// Mitsubishi GX Works2 project: PuyoPuyo_Ver100_20220530   PLC: Q03UDV

PROGRAM 11_DEBUG  // Test Function for Debug
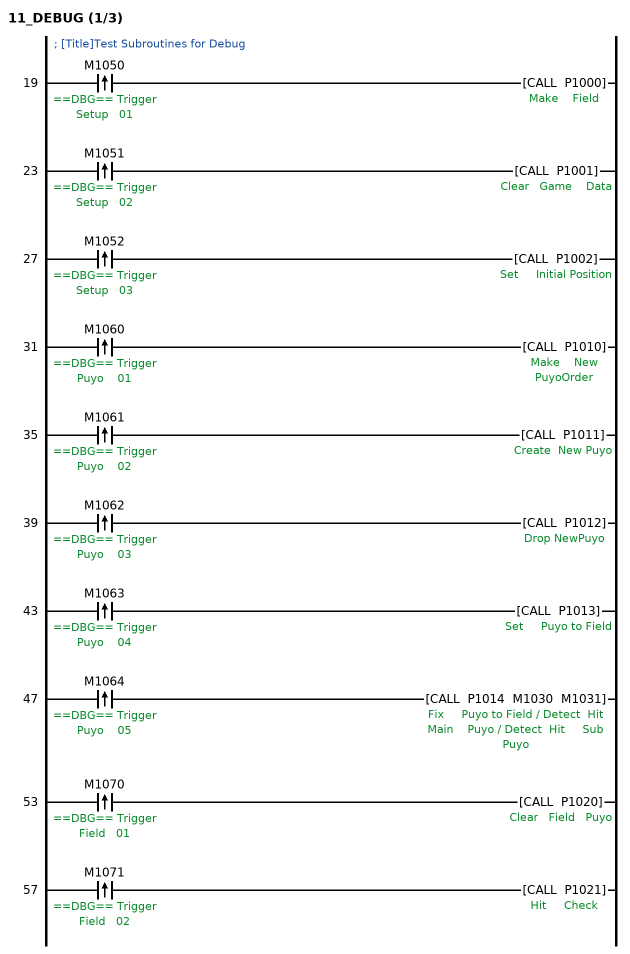
; [Title]Test Subroutines for Debug
19    LDP     M1050  ; ==DBG== Trigger Setup   01
      CALL    P1000  ; Make    Field
23    LDP     M1051  ; ==DBG== Trigger Setup   02
      CALL    P1001  ; Clear   Game    Data
27    LDP     M1052  ; ==DBG== Trigger Setup   03
      CALL    P1002  ; Set     Initial Position
31    LDP     M1060  ; ==DBG== Trigger Puyo    01
      CALL    P1010  ; Make    New PuyoOrder
35    LDP     M1061  ; ==DBG== Trigger Puyo    02
      CALL    P1011  ; Create  New Puyo
39    LDP     M1062  ; ==DBG== Trigger Puyo    03
      CALL    P1012  ; Drop NewPuyo
43    LDP     M1063  ; ==DBG== Trigger Puyo    04
      CALL    P1013  ; Set     Puyo to Field
47    LDP     M1064  ; ==DBG== Trigger Puyo    05
      CALL    P1014 M1030 M1031  ; Fix     Puyo to Field / Detect  Hit     Main    Puyo / Detect  Hit     Sub     Puyo
53    LDP     M1070  ; ==DBG== Trigger Field   01
      CALL    P1020  ; Clear   Field   Puyo
57    LDP     M1071  ; ==DBG== Trigger Field   02
      CALL    P1021  ; Hit     Check
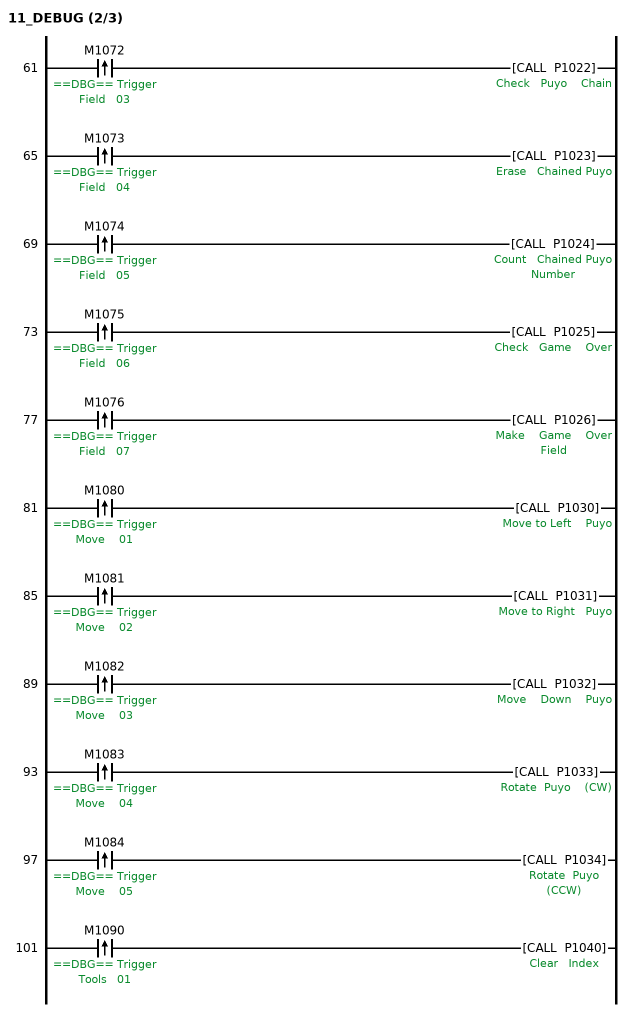
61    LDP     M1072  ; ==DBG== Trigger Field   03
      CALL    P1022  ; Check   Puyo    Chain
65    LDP     M1073  ; ==DBG== Trigger Field   04
      CALL    P1023  ; Erase   Chained Puyo
69    LDP     M1074  ; ==DBG== Trigger Field   05
      CALL    P1024  ; Count   Chained Puyo    Number
73    LDP     M1075  ; ==DBG== Trigger Field   06
      CALL    P1025  ; Check   Game    Over
77    LDP     M1076  ; ==DBG== Trigger Field   07
      CALL    P1026  ; Make    Game    Over    Field
81    LDP     M1080  ; ==DBG== Trigger Move    01
      CALL    P1030  ; Move to Left    Puyo
85    LDP     M1081  ; ==DBG== Trigger Move    02
      CALL    P1031  ; Move to Right   Puyo
89    LDP     M1082  ; ==DBG== Trigger Move    03
      CALL    P1032  ; Move    Down    Puyo
93    LDP     M1083  ; ==DBG== Trigger Move    04
      CALL    P1033  ; Rotate  Puyo    (CW)
97    LDP     M1084  ; ==DBG== Trigger Move    05
      CALL    P1034  ; Rotate  Puyo    (CCW)
101   LDP     M1090  ; ==DBG== Trigger Tools   01
      CALL    P1040  ; Clear   Index
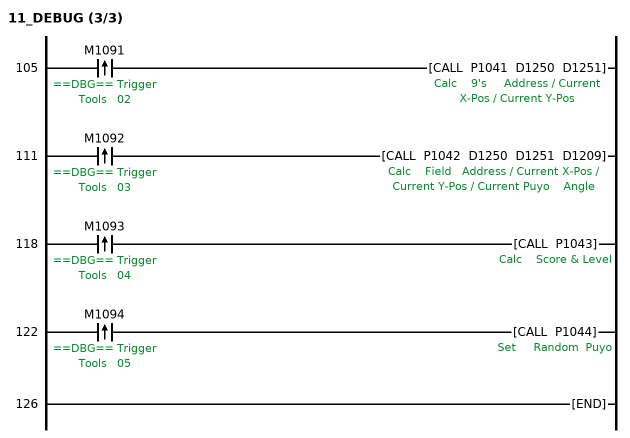
105   LDP     M1091  ; ==DBG== Trigger Tools   02
      CALL    P1041 D1250 D1251  ; Calc    9's     Address / Current X-Pos / Current Y-Pos
111   LDP     M1092  ; ==DBG== Trigger Tools   03
      CALL    P1042 D1250 D1251 D1209  ; Calc    Field   Address / Current Puyo    Angle
118   LDP     M1093  ; ==DBG== Trigger Tools   04
      CALL    P1043  ; Calc    Score & Level
122   LDP     M1094  ; ==DBG== Trigger Tools   05
      CALL    P1044  ; Set     Random  Puyo
126   END
END_PROGRAM

PROGRAM 95_TOOL  // Common Tools
; [Title]P1040 Clear Index
      P1040
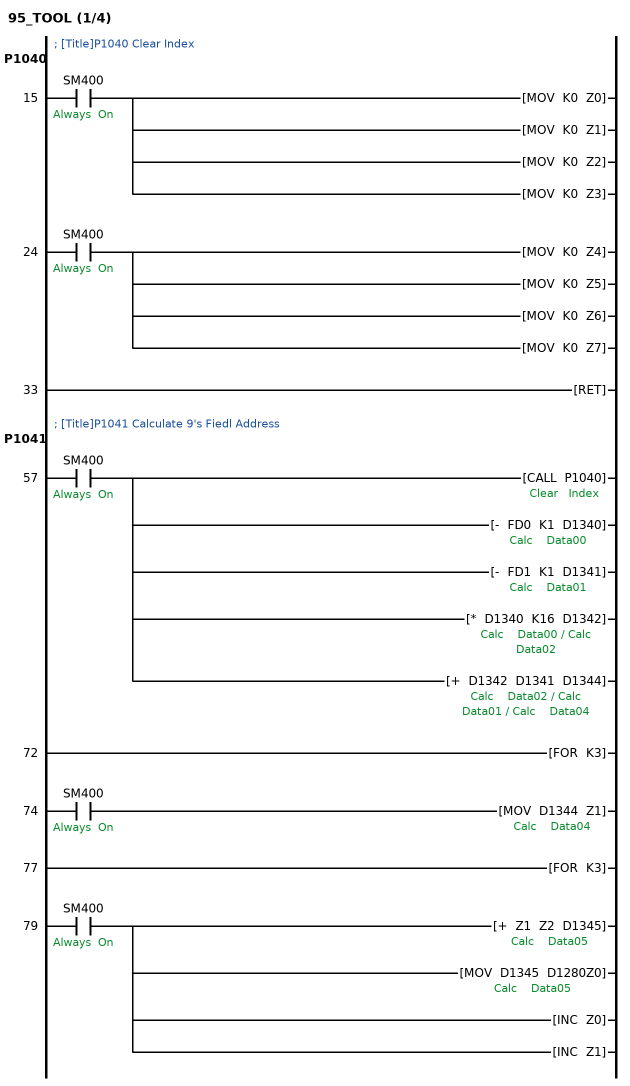
15    LD      SM400  ; Always  On
      MOV     K0 Z0
      MOV     K0 Z1
      MOV     K0 Z2
      MOV     K0 Z3
24    LD      SM400  ; Always  On
      MOV     K0 Z4
      MOV     K0 Z5
      MOV     K0 Z6
      MOV     K0 Z7
33    RET
; [Title]P1041 Calculate 9's Fiedl Address
      P1041
57    LD      SM400  ; Always  On
      CALL    P1040  ; Clear   Index
      -       FD0 K1 D1340  ; Calc    Data00
      -       FD1 K1 D1341  ; Calc    Data01
      *       D1340 K16 D1342  ; Calc    Data02
      +       D1342 D1341 D1344  ; Calc    Data04
72    FOR     K3
74    LD      SM400  ; Always  On
      MOV     D1344 Z1
77    FOR     K3
79    LD      SM400  ; Always  On
      +       Z1 Z2 D1345  ; Calc    Data05
      MOV     D1345 D1280Z0
      INC     Z0
      INC     Z1
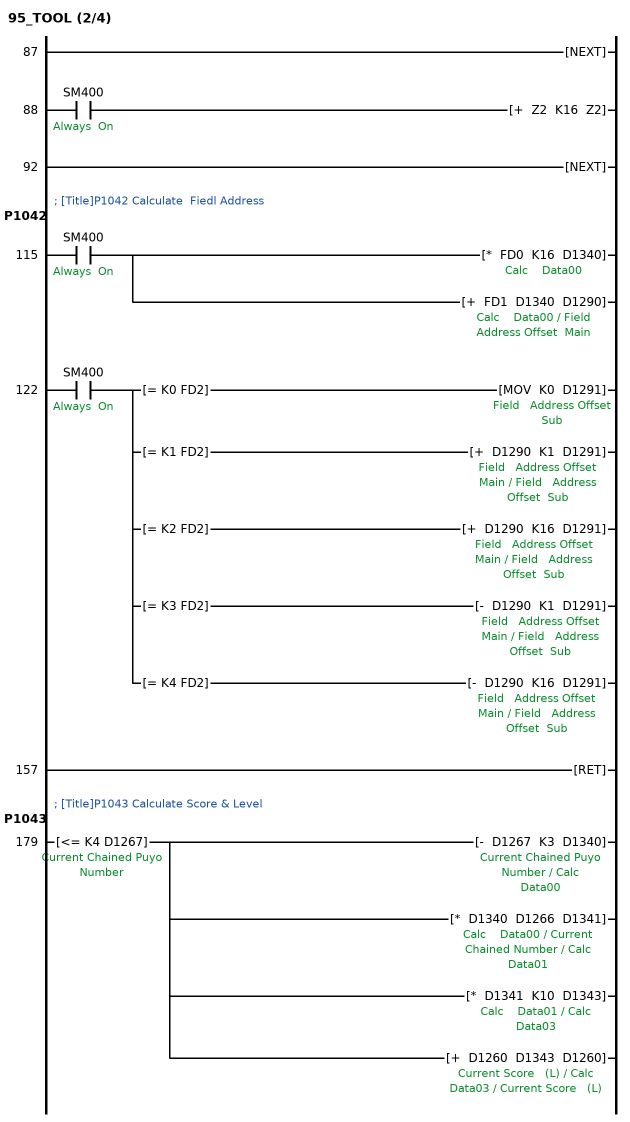
87    NEXT
88    LD      SM400  ; Always  On
      +       Z2 K16 Z2
92    NEXT
; [Title]P1042 Calculate  Fiedl Address
      P1042
115   LD      SM400  ; Always  On
      *       FD0 K16 D1340
      +       FD1 D1340 D1290  ; Field   Address Offset  Main
122   LD      SM400  ; Always  On
      MPS
      AND=    K0 FD2
      MOV     K0 D1291  ; Field   Address Offset  Sub
      MRD
      AND=    K1 FD2
      +       D1290 K1 D1291
      MRD
      AND=    K2 FD2
      +       D1290 K16 D1291
      MRD
      AND=    K3 FD2
      -       D1290 K1 D1291
      MPP
      AND=    K4 FD2
      -       D1290 K16 D1291
157   RET
; [Title]P1043 Calculate Score & Level
      P1043
179   LD<=    K4 D1267  ; Current Chained Puyo    Number
      -       D1267 K3 D1340
      *       D1340 D1266 D1341  ; Current Chained Number
      *       D1341 K10 D1343  ; Calc    Data03
      +       D1260 D1343 D1260  ; Current Score   (L)
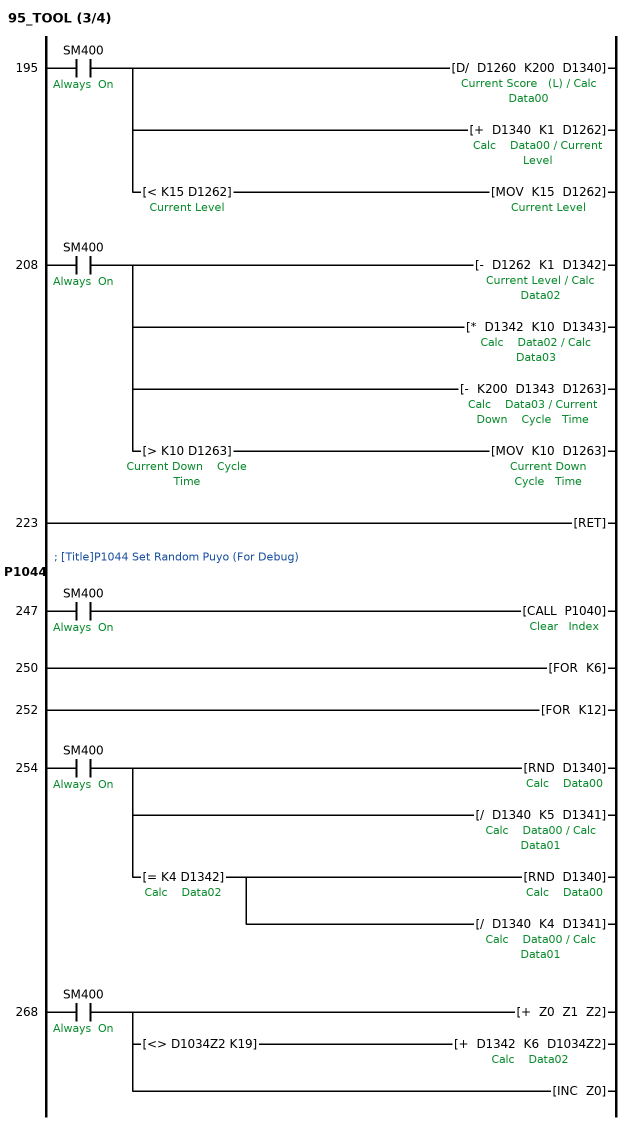
195   LD      SM400  ; Always  On
      D/      D1260 K200 D1340
      +       D1340 K1 D1262  ; Current Level
      AND<    K15 D1262  ; Current Level
      MOV     K15 D1262
208   LD      SM400  ; Always  On
      -       D1262 K1 D1342
      *       D1342 K10 D1343
      -       K200 D1343 D1263  ; Current Down    Cycle   Time
      AND>    K10 D1263  ; Current Down    Cycle   Time
      MOV     K10 D1263
223   RET
; [Title]P1044 Set Random Puyo (For Debug)
      P1044
247   LD      SM400  ; Always  On
      CALL    P1040
250   FOR     K6
252   FOR     K12
254   LD      SM400  ; Always  On
      RND     D1340
      /       D1340 K5 D1341
      AND=    K4 D1342  ; Calc    Data02
      RND     D1340
      /       D1340 K4 D1341
268   LD      SM400  ; Always  On
      +       Z0 Z1 Z2
      MPS
      AND<>   D1034Z2 K19
      +       D1342 K6 D1034Z2
      MPP
      INC     Z0
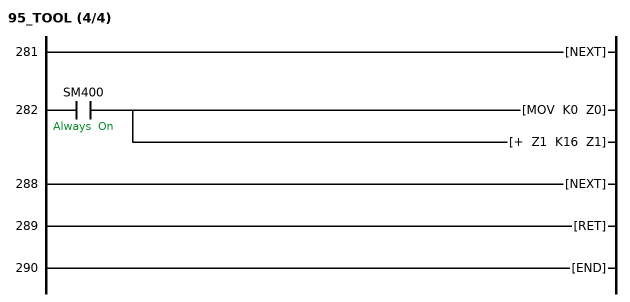
281   NEXT
282   LD      SM400  ; Always  On
      MOV     K0 Z0
      +       Z1 K16 Z1
288   NEXT
289   RET
290   END
END_PROGRAM

PROGRAM 91_SETUP  // Setup Condition
; [Title]P1000 Make Field
; Field Data K0 = Blank(No Puyo), K19 = Wall
      P1000
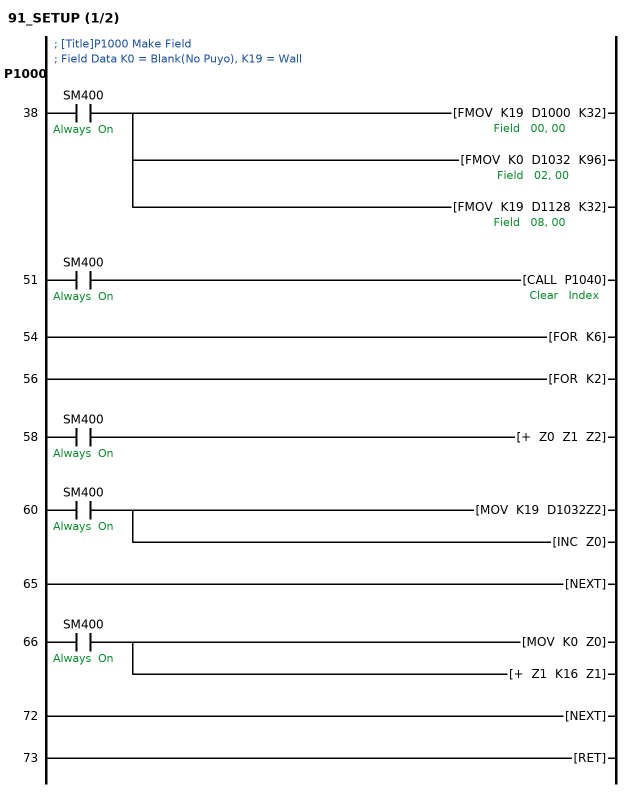
38    LD      SM400  ; Always  On
      FMOV    K19 D1000 K32  ; Field   00, 00
      FMOV    K0 D1032 K96  ; Field   02, 00
      FMOV    K19 D1128 K32  ; Field   08, 00
51    LD      SM400  ; Always  On
      CALL    P1040  ; Clear   Index
54    FOR     K6
56    FOR     K2
58    LD      SM400  ; Always  On
      +       Z0 Z1 Z2
60    LD      SM400  ; Always  On
      MOV     K19 D1032Z2
      INC     Z0
65    NEXT
66    LD      SM400  ; Always  On
      MOV     K0 Z0
      +       Z1 K16 Z1
72    NEXT
73    RET
; [Title]P1001 Clear All Game Data
      P1001
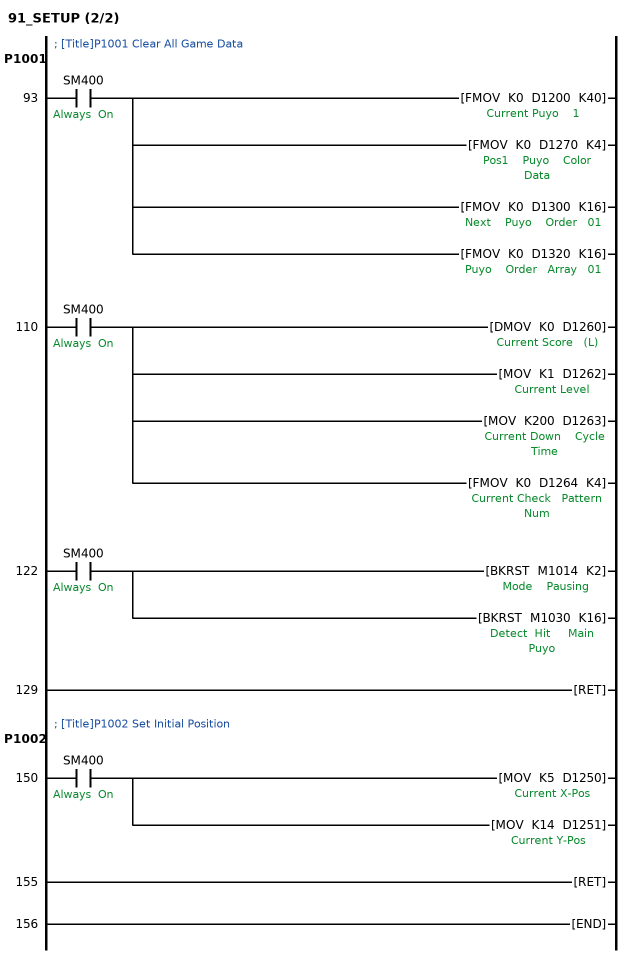
93    LD      SM400  ; Always  On
      FMOV    K0 D1200 K40  ; Current Puyo    1
      FMOV    K0 D1270 K4  ; Pos1    Puyo    Color   Data
      FMOV    K0 D1300 K16  ; Next    Puyo    Order   01
      FMOV    K0 D1320 K16  ; Puyo    Order   Array   01
110   LD      SM400  ; Always  On
      DMOV    K0 D1260  ; Current Score   (L)
      MOV     K1 D1262  ; Current Level
      MOV     K200 D1263  ; Current Down    Cycle   Time
      FMOV    K0 D1264 K4  ; Current Check   Pattern Num
122   LD      SM400  ; Always  On
      BKRST   M1014 K2  ; Mode    Pausing
      BKRST   M1030 K16  ; Detect  Hit     Main    Puyo
129   RET
; [Title]P1002 Set Initial Position
      P1002
150   LD      SM400  ; Always  On
      MOV     K5 D1250  ; Current X-Pos
      MOV     K14 D1251  ; Current Y-Pos
155   RET
156   END
END_PROGRAM

PROGRAM 01_INIT  // Initializing Data
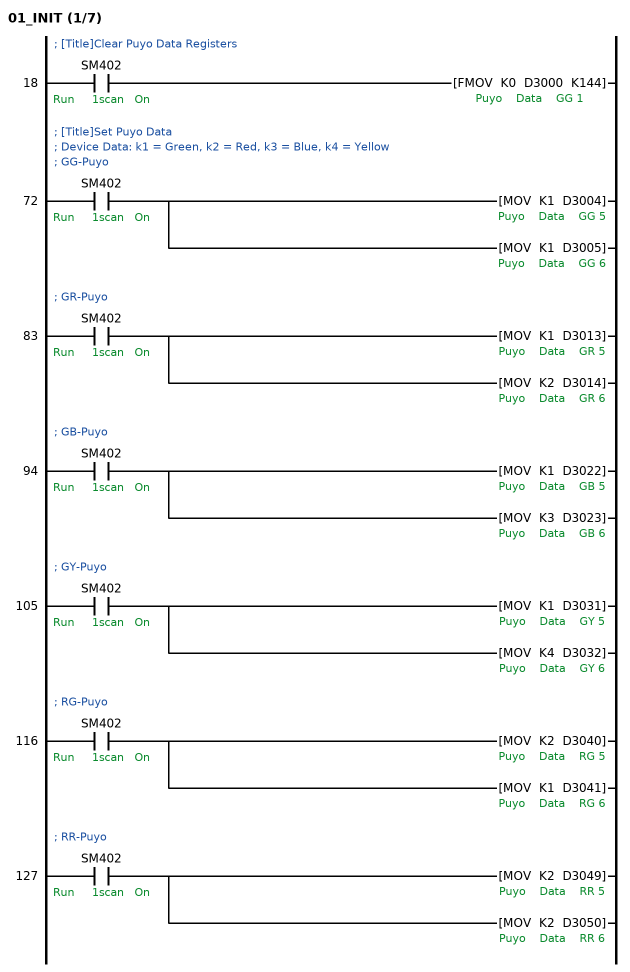
; [Title]Clear Puyo Data Registers
18    LD      SM402  ; Run     1scan   On
      FMOV    K0 D3000 K144  ; Puyo    Data    GG 1
; [Title]Set Puyo Data
; Device Data: k1 = Green, k2 = Red, k3 = Blue, k4 = Yellow
; GG-Puyo
72    LD      SM402  ; Run     1scan   On
      MOV     K1 D3004  ; Puyo    Data    GG 5
      MOV     K1 D3005  ; Puyo    Data    GG 6
; GR-Puyo
83    LD      SM402  ; Run     1scan   On
      MOV     K1 D3013  ; Puyo    Data    GR 5
      MOV     K2 D3014  ; Puyo    Data    GR 6
; GB-Puyo
94    LD      SM402  ; Run     1scan   On
      MOV     K1 D3022  ; Puyo    Data    GB 5
      MOV     K3 D3023  ; Puyo    Data    GB 6
; GY-Puyo
105   LD      SM402  ; Run     1scan   On
      MOV     K1 D3031  ; Puyo    Data    GY 5
      MOV     K4 D3032  ; Puyo    Data    GY 6
; RG-Puyo
116   LD      SM402  ; Run     1scan   On
      MOV     K2 D3040  ; Puyo    Data    RG 5
      MOV     K1 D3041  ; Puyo    Data    RG 6
; RR-Puyo
127   LD      SM402  ; Run     1scan   On
      MOV     K2 D3049  ; Puyo    Data    RR 5
      MOV     K2 D3050  ; Puyo    Data    RR 6
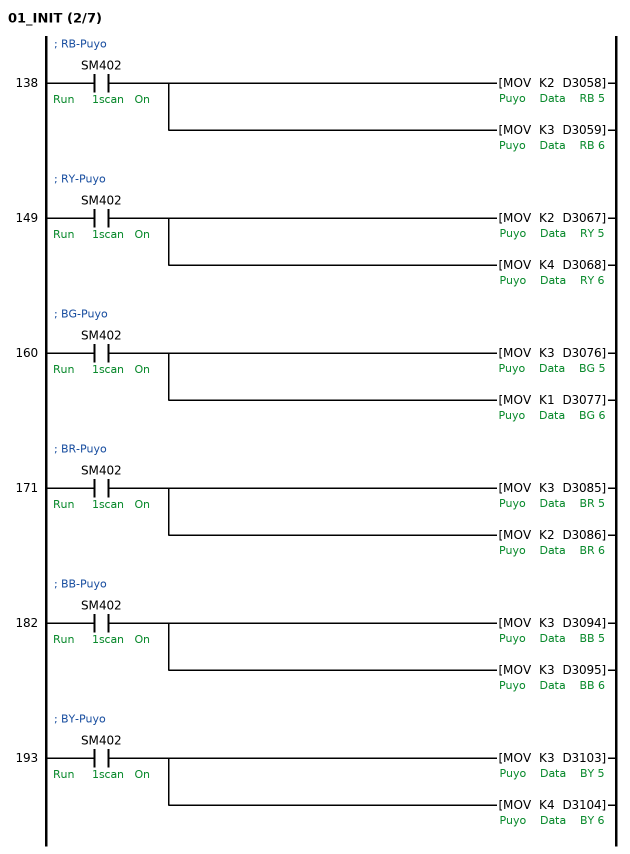
; RB-Puyo
138   LD      SM402  ; Run     1scan   On
      MOV     K2 D3058  ; Puyo    Data    RB 5
      MOV     K3 D3059  ; Puyo    Data    RB 6
; RY-Puyo
149   LD      SM402  ; Run     1scan   On
      MOV     K2 D3067  ; Puyo    Data    RY 5
      MOV     K4 D3068  ; Puyo    Data    RY 6
; BG-Puyo
160   LD      SM402  ; Run     1scan   On
      MOV     K3 D3076  ; Puyo    Data    BG 5
      MOV     K1 D3077  ; Puyo    Data    BG 6
; BR-Puyo
171   LD      SM402  ; Run     1scan   On
      MOV     K3 D3085  ; Puyo    Data    BR 5
      MOV     K2 D3086  ; Puyo    Data    BR 6
; BB-Puyo
182   LD      SM402  ; Run     1scan   On
      MOV     K3 D3094  ; Puyo    Data    BB 5
      MOV     K3 D3095  ; Puyo    Data    BB 6
; BY-Puyo
193   LD      SM402  ; Run     1scan   On
      MOV     K3 D3103  ; Puyo    Data    BY 5
      MOV     K4 D3104  ; Puyo    Data    BY 6
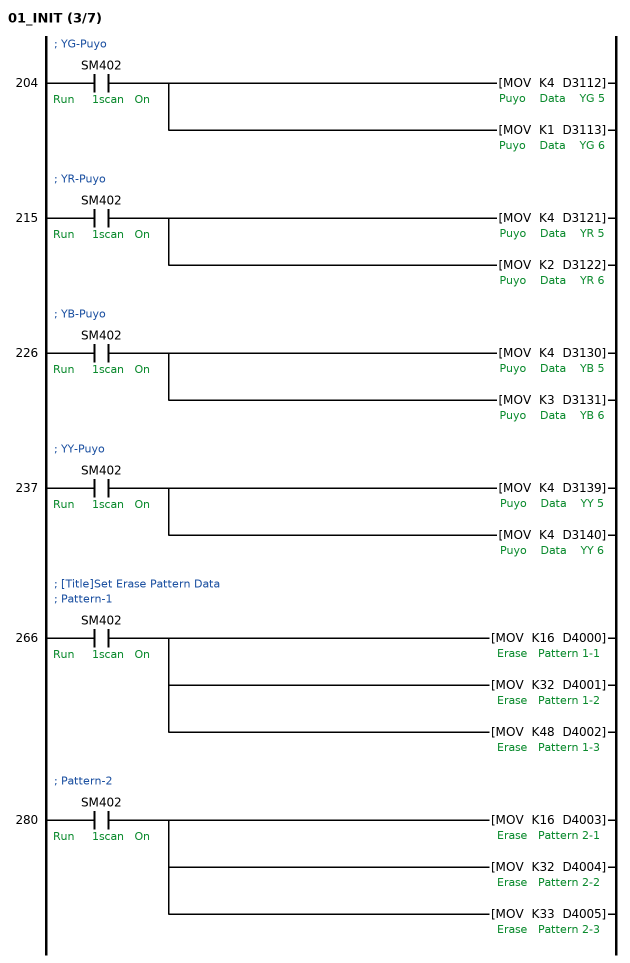
; YG-Puyo
204   LD      SM402  ; Run     1scan   On
      MOV     K4 D3112  ; Puyo    Data    YG 5
      MOV     K1 D3113  ; Puyo    Data    YG 6
; YR-Puyo
215   LD      SM402  ; Run     1scan   On
      MOV     K4 D3121  ; Puyo    Data    YR 5
      MOV     K2 D3122  ; Puyo    Data    YR 6
; YB-Puyo
226   LD      SM402  ; Run     1scan   On
      MOV     K4 D3130  ; Puyo    Data    YB 5
      MOV     K3 D3131  ; Puyo    Data    YB 6
; YY-Puyo
237   LD      SM402  ; Run     1scan   On
      MOV     K4 D3139  ; Puyo    Data    YY 5
      MOV     K4 D3140  ; Puyo    Data    YY 6
; [Title]Set Erase Pattern Data
; Pattern-1
266   LD      SM402  ; Run     1scan   On
      MOV     K16 D4000  ; Erase   Pattern 1-1
      MOV     K32 D4001  ; Erase   Pattern 1-2
      MOV     K48 D4002  ; Erase   Pattern 1-3
; Pattern-2
280   LD      SM402  ; Run     1scan   On
      MOV     K16 D4003  ; Erase   Pattern 2-1
      MOV     K32 D4004  ; Erase   Pattern 2-2
      MOV     K33 D4005  ; Erase   Pattern 2-3
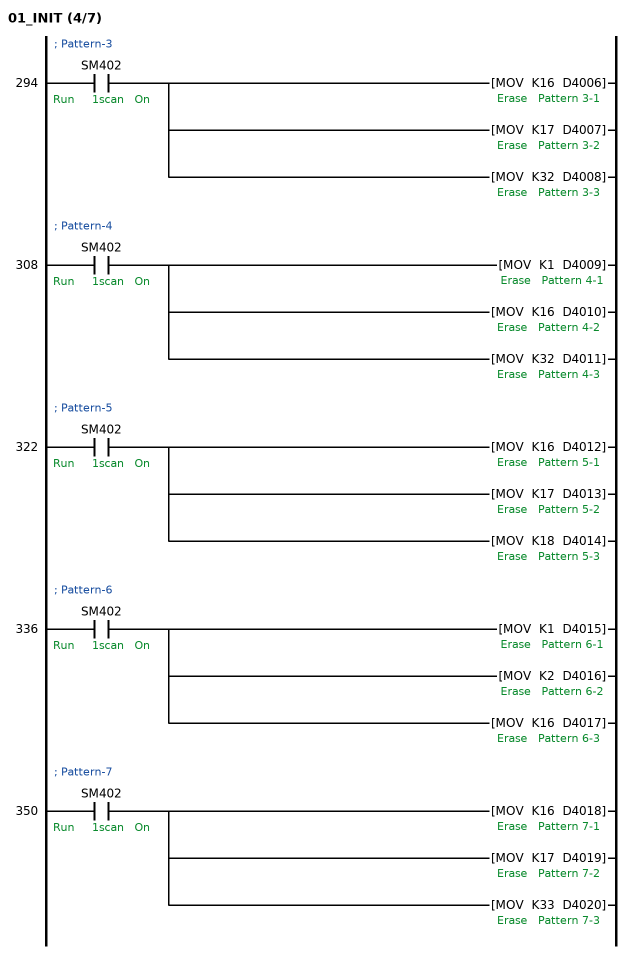
; Pattern-3
294   LD      SM402  ; Run     1scan   On
      MOV     K16 D4006  ; Erase   Pattern 3-1
      MOV     K17 D4007  ; Erase   Pattern 3-2
      MOV     K32 D4008  ; Erase   Pattern 3-3
; Pattern-4
308   LD      SM402  ; Run     1scan   On
      MOV     K1 D4009  ; Erase   Pattern 4-1
      MOV     K16 D4010  ; Erase   Pattern 4-2
      MOV     K32 D4011  ; Erase   Pattern 4-3
; Pattern-5
322   LD      SM402  ; Run     1scan   On
      MOV     K16 D4012  ; Erase   Pattern 5-1
      MOV     K17 D4013  ; Erase   Pattern 5-2
      MOV     K18 D4014  ; Erase   Pattern 5-3
; Pattern-6
336   LD      SM402  ; Run     1scan   On
      MOV     K1 D4015  ; Erase   Pattern 6-1
      MOV     K2 D4016  ; Erase   Pattern 6-2
      MOV     K16 D4017  ; Erase   Pattern 6-3
; Pattern-7
350   LD      SM402  ; Run     1scan   On
      MOV     K16 D4018  ; Erase   Pattern 7-1
      MOV     K17 D4019  ; Erase   Pattern 7-2
      MOV     K33 D4020  ; Erase   Pattern 7-3
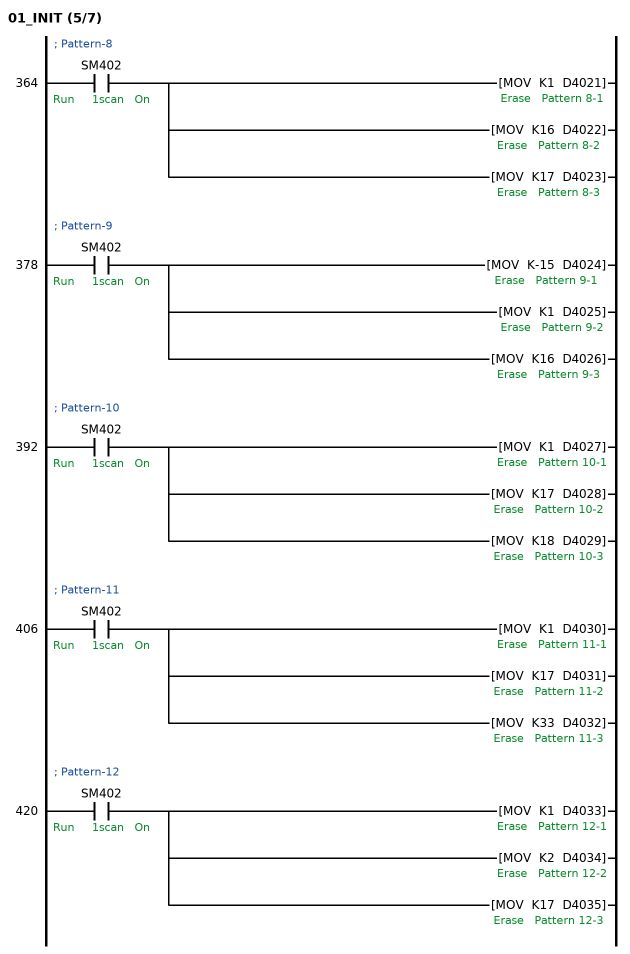
; Pattern-8
364   LD      SM402  ; Run     1scan   On
      MOV     K1 D4021  ; Erase   Pattern 8-1
      MOV     K16 D4022  ; Erase   Pattern 8-2
      MOV     K17 D4023  ; Erase   Pattern 8-3
; Pattern-9
378   LD      SM402  ; Run     1scan   On
      MOV     K-15 D4024  ; Erase   Pattern 9-1
      MOV     K1 D4025  ; Erase   Pattern 9-2
      MOV     K16 D4026  ; Erase   Pattern 9-3
; Pattern-10
392   LD      SM402  ; Run     1scan   On
      MOV     K1 D4027  ; Erase   Pattern 10-1
      MOV     K17 D4028  ; Erase   Pattern 10-2
      MOV     K18 D4029  ; Erase   Pattern 10-3
; Pattern-11
406   LD      SM402  ; Run     1scan   On
      MOV     K1 D4030  ; Erase   Pattern 11-1
      MOV     K17 D4031  ; Erase   Pattern 11-2
      MOV     K33 D4032  ; Erase   Pattern 11-3
; Pattern-12
420   LD      SM402  ; Run     1scan   On
      MOV     K1 D4033  ; Erase   Pattern 12-1
      MOV     K2 D4034  ; Erase   Pattern 12-2
      MOV     K17 D4035  ; Erase   Pattern 12-3
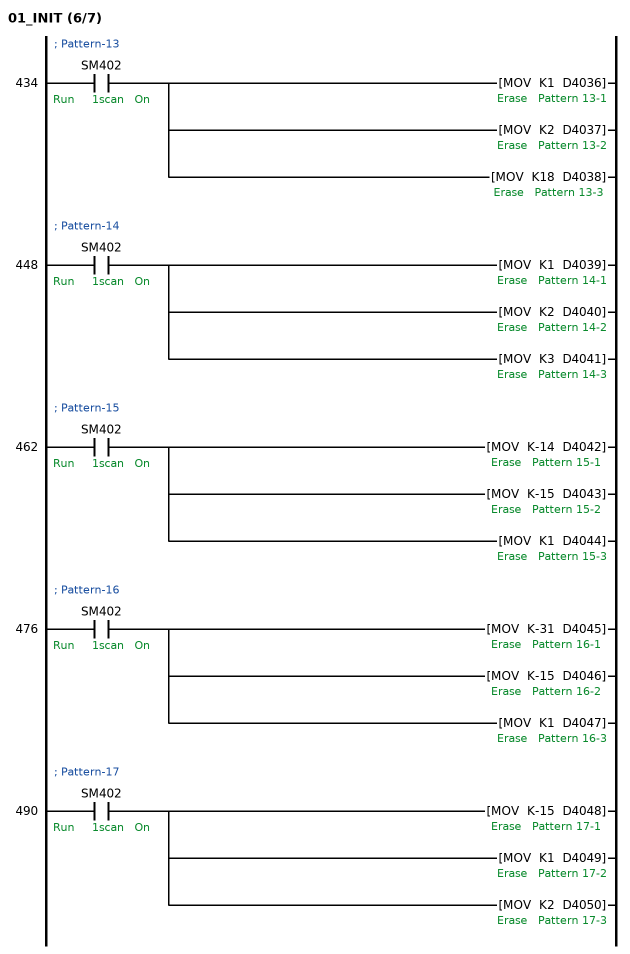
; Pattern-13
434   LD      SM402  ; Run     1scan   On
      MOV     K1 D4036  ; Erase   Pattern 13-1
      MOV     K2 D4037  ; Erase   Pattern 13-2
      MOV     K18 D4038  ; Erase   Pattern 13-3
; Pattern-14
448   LD      SM402  ; Run     1scan   On
      MOV     K1 D4039  ; Erase   Pattern 14-1
      MOV     K2 D4040  ; Erase   Pattern 14-2
      MOV     K3 D4041  ; Erase   Pattern 14-3
; Pattern-15
462   LD      SM402  ; Run     1scan   On
      MOV     K-14 D4042  ; Erase   Pattern 15-1
      MOV     K-15 D4043  ; Erase   Pattern 15-2
      MOV     K1 D4044  ; Erase   Pattern 15-3
; Pattern-16
476   LD      SM402  ; Run     1scan   On
      MOV     K-31 D4045  ; Erase   Pattern 16-1
      MOV     K-15 D4046  ; Erase   Pattern 16-2
      MOV     K1 D4047  ; Erase   Pattern 16-3
; Pattern-17
490   LD      SM402  ; Run     1scan   On
      MOV     K-15 D4048  ; Erase   Pattern 17-1
      MOV     K1 D4049  ; Erase   Pattern 17-2
      MOV     K2 D4050  ; Erase   Pattern 17-3
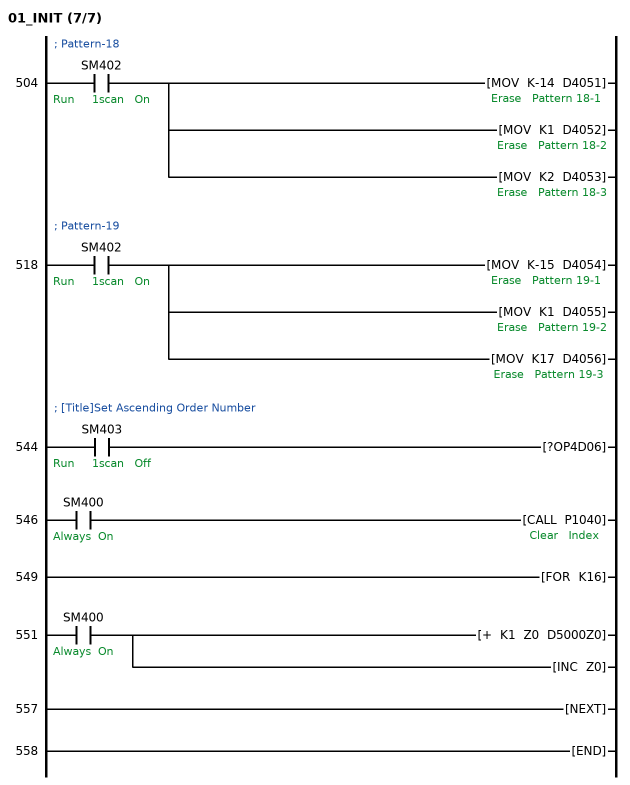
; Pattern-18
504   LD      SM402  ; Run     1scan   On
      MOV     K-14 D4051  ; Erase   Pattern 18-1
      MOV     K1 D4052  ; Erase   Pattern 18-2
      MOV     K2 D4053  ; Erase   Pattern 18-3
; Pattern-19
518   LD      SM402  ; Run     1scan   On
      MOV     K-15 D4054  ; Erase   Pattern 19-1
      MOV     K1 D4055  ; Erase   Pattern 19-2
      MOV     K17 D4056  ; Erase   Pattern 19-3
; [Title]Set Ascending Order Number
544   LD      SM403  ; Run     1scan   Off
      ?OP4D06
546   LD      SM400  ; Always  On
      CALL    P1040  ; Clear   Index
549   FOR     K16
551   LD      SM400  ; Always  On
      +       K1 Z0 D5000Z0
      INC     Z0
557   NEXT
558   END
END_PROGRAM

PROGRAM 92_PUYO  // Set Puyo Data
; [Title]P1010 Make New Puyo Order
      P1010
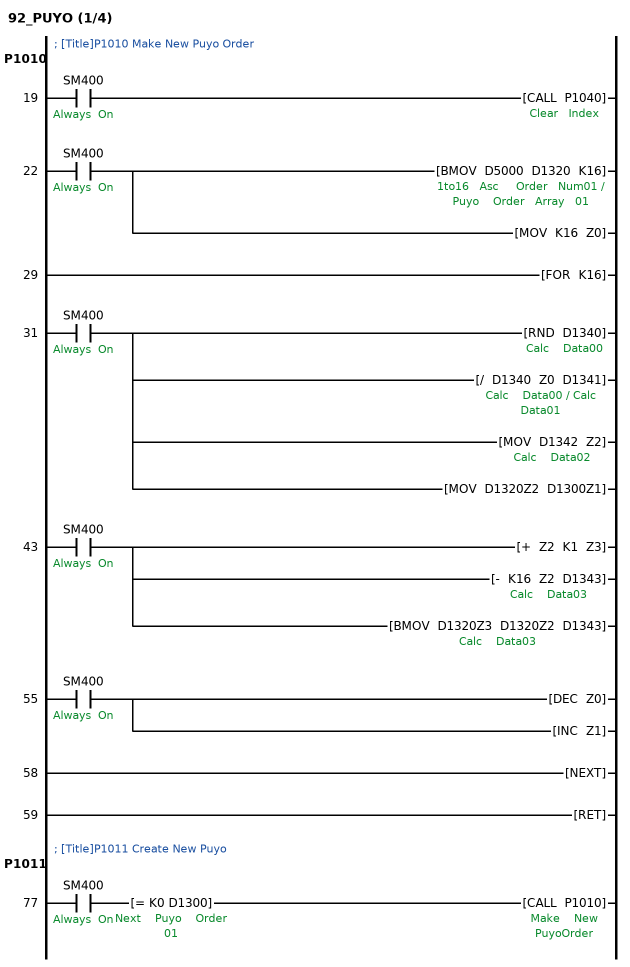
19    LD      SM400  ; Always  On
      CALL    P1040  ; Clear   Index
22    LD      SM400  ; Always  On
      BMOV    D5000 D1320 K16  ; 1to16   Asc     Order   Num01 / Puyo    Order   Array   01
      MOV     K16 Z0
29    FOR     K16
31    LD      SM400  ; Always  On
      RND     D1340  ; Calc    Data00
      /       D1340 Z0 D1341  ; Calc    Data01
      MOV     D1342 Z2  ; Calc    Data02
      MOV     D1320Z2 D1300Z1
43    LD      SM400  ; Always  On
      +       Z2 K1 Z3
      -       K16 Z2 D1343  ; Calc    Data03
      BMOV    D1320Z3 D1320Z2 D1343
55    LD      SM400  ; Always  On
      DEC     Z0
      INC     Z1
58    NEXT
59    RET
; [Title]P1011 Create New Puyo
      P1011
77    LD      SM400  ; Always  On
      AND=    K0 D1300  ; Next    Puyo    Order   01
      CALL    P1010  ; Make    New PuyoOrder
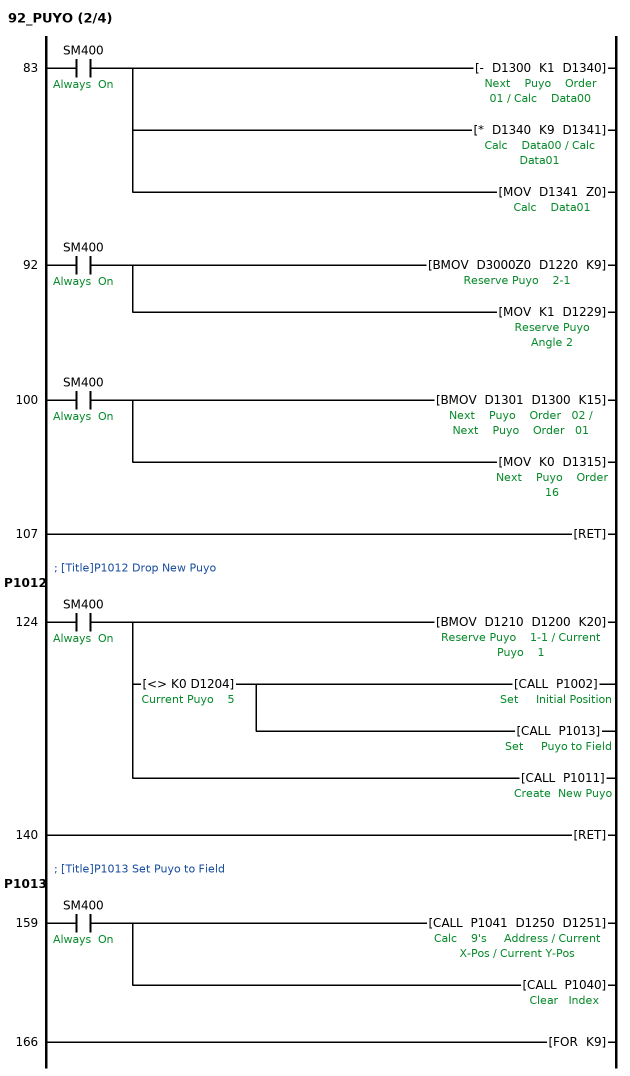
83    LD      SM400  ; Always  On
      -       D1300 K1 D1340
      *       D1340 K9 D1341
      MOV     D1341 Z0
92    LD      SM400  ; Always  On
      BMOV    D3000Z0 D1220 K9  ; Reserve Puyo    2-1
      MOV     K1 D1229  ; Reserve Puyo    Angle 2
100   LD      SM400  ; Always  On
      BMOV    D1301 D1300 K15  ; Next    Puyo    Order   02
      MOV     K0 D1315  ; Next    Puyo    Order   16
107   RET
; [Title]P1012 Drop New Puyo
      P1012
124   LD      SM400  ; Always  On
      BMOV    D1210 D1200 K20  ; Reserve Puyo    1-1 / Current Puyo    1
      MPS
      AND<>   K0 D1204  ; Current Puyo    5
      CALL    P1002  ; Set     Initial Position
      CALL    P1013  ; Set     Puyo to Field
      MPP
      CALL    P1011  ; Create  New Puyo
140   RET
; [Title]P1013 Set Puyo to Field
      P1013
159   LD      SM400  ; Always  On
      CALL    P1041 D1250 D1251  ; Calc    9's     Address / Current X-Pos / Current Y-Pos
      CALL    P1040
166   FOR     K9
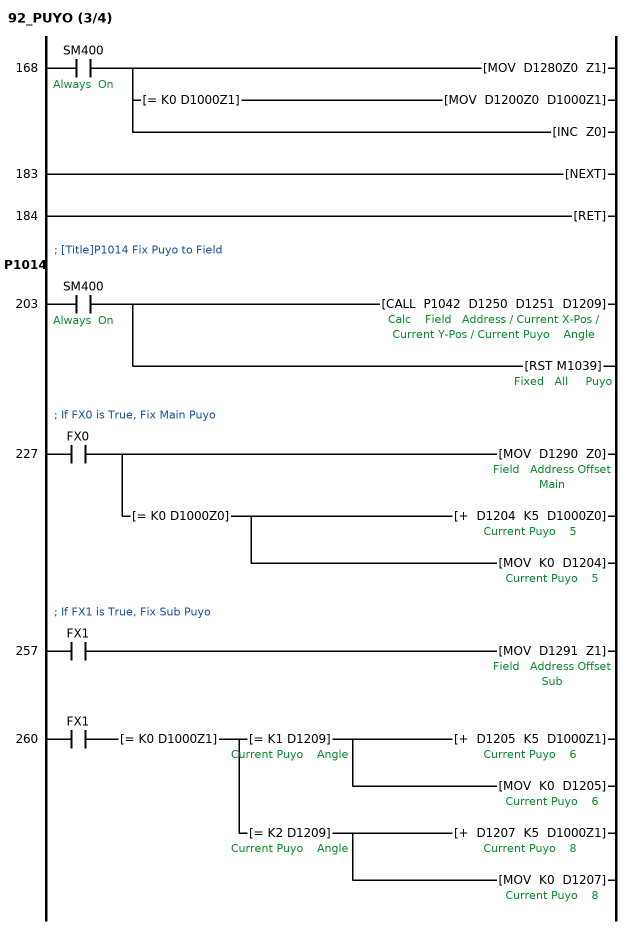
168   LD      SM400  ; Always  On
      MOV     D1280Z0 Z1
      MPS
      AND=    K0 D1000Z1
      MOV     D1200Z0 D1000Z1
      MPP
      INC     Z0
183   NEXT
184   RET
; [Title]P1014 Fix Puyo to Field
      P1014
203   LD      SM400  ; Always  On
      CALL    P1042 D1250 D1251 D1209  ; Calc    Field   Address / Current Puyo    Angle
      RST     M1039  ; Fixed   All     Puyo
; If FX0 is True, Fix Main Puyo
227   LD      FX0
      MOV     D1290 Z0  ; Field   Address Offset  Main
      AND=    K0 D1000Z0
      +       D1204 K5 D1000Z0
      MOV     K0 D1204
; If FX1 is True, Fix Sub Puyo
257   LD      FX1
      MOV     D1291 Z1  ; Field   Address Offset  Sub
260   LD      FX1
      AND=    K0 D1000Z1
      MPS
      AND=    K1 D1209  ; Current Puyo    Angle
      +       D1205 K5 D1000Z1  ; Current Puyo    6
      MOV     K0 D1205
      MPP
      AND=    K2 D1209  ; Current Puyo    Angle
      +       D1207 K5 D1000Z1  ; Current Puyo    8
      MOV     K0 D1207
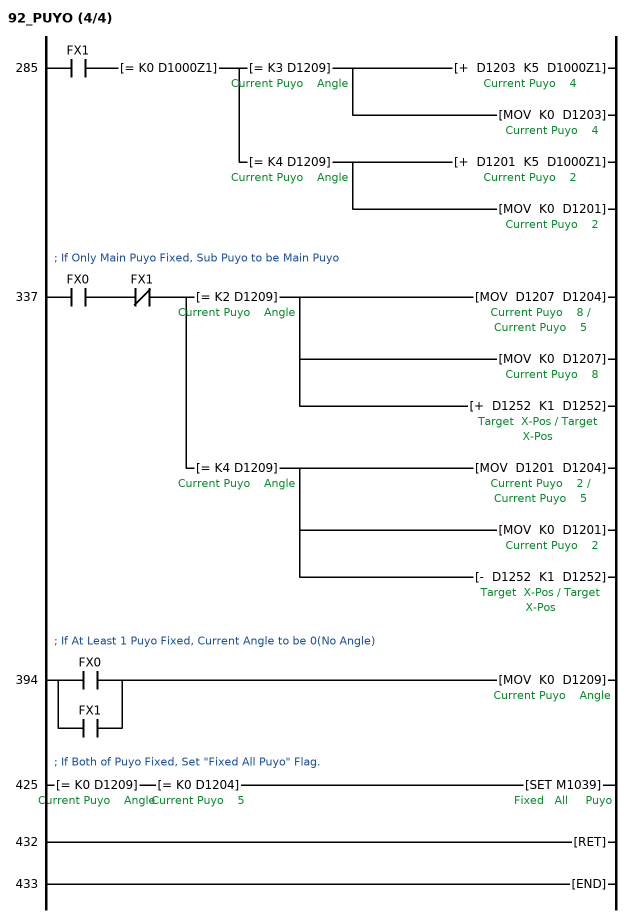
285   LD      FX1
      AND=    K0 D1000Z1
      MPS
      AND=    K3 D1209  ; Current Puyo    Angle
      +       D1203 K5 D1000Z1  ; Current Puyo    4
      MOV     K0 D1203
      MPP
      AND=    K4 D1209  ; Current Puyo    Angle
      +       D1201 K5 D1000Z1  ; Current Puyo    2
      MOV     K0 D1201
; If Only Main Puyo Fixed, Sub Puyo to be Main Puyo
337   LD      FX0
      ANI     FX1
      MPS
      AND=    K2 D1209  ; Current Puyo    Angle
      MOV     D1207 D1204
      MOV     K0 D1207
      +       D1252 K1 D1252  ; Target  X-Pos
      MPP
      AND=    K4 D1209  ; Current Puyo    Angle
      MOV     D1201 D1204
      MOV     K0 D1201
      -       D1252 K1 D1252
; If At Least 1 Puyo Fixed, Current Angle to be 0(No Angle)
394   LD      FX0
      OR      FX1
      MOV     K0 D1209
; If Both of Puyo Fixed, Set "Fixed All Puyo" Flag.
425   LD=     K0 D1209  ; Current Puyo    Angle
      AND=    K0 D1204  ; Current Puyo    5
      SET     M1039  ; Fixed   All     Puyo
432   RET
433   END
END_PROGRAM

PROGRAM 93_FIELD  // Manage Field
; [Title]P1020 Clear Field Puyo
      P1020
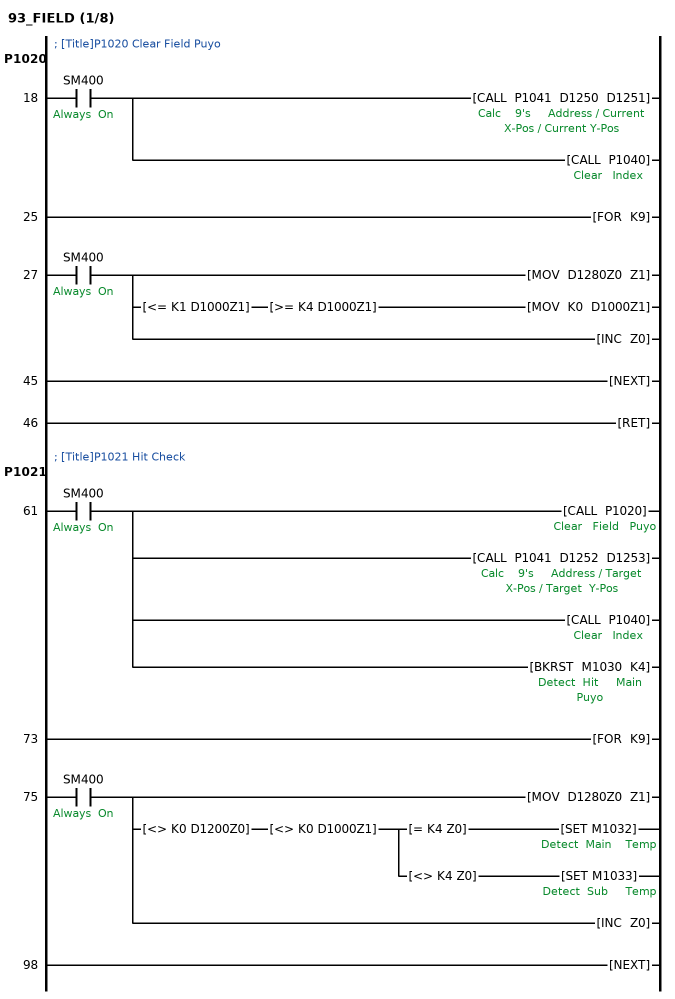
18    LD      SM400  ; Always  On
      CALL    P1041 D1250 D1251  ; Calc    9's     Address / Current X-Pos / Current Y-Pos
      CALL    P1040  ; Clear   Index
25    FOR     K9
27    LD      SM400  ; Always  On
      MOV     D1280Z0 Z1
      MPS
      AND<=   K1 D1000Z1
      AND>=   K4 D1000Z1
      MOV     K0 D1000Z1
      MPP
      INC     Z0
45    NEXT
46    RET
; [Title]P1021 Hit Check
      P1021
61    LD      SM400  ; Always  On
      CALL    P1020  ; Clear   Field   Puyo
      CALL    P1041 D1252 D1253  ; Target  X-Pos / Target  Y-Pos
      CALL    P1040
      BKRST   M1030 K4  ; Detect  Hit     Main    Puyo
73    FOR     K9
75    LD      SM400  ; Always  On
      MOV     D1280Z0 Z1
      MPS
      AND<>   K0 D1200Z0
      AND<>   K0 D1000Z1
      MPS
      AND=    K4 Z0
      SET     M1032  ; Detect  Main    Temp
      MPP
      AND<>   K4 Z0
      SET     M1033  ; Detect  Sub     Temp
      MPP
      INC     Z0
98    NEXT
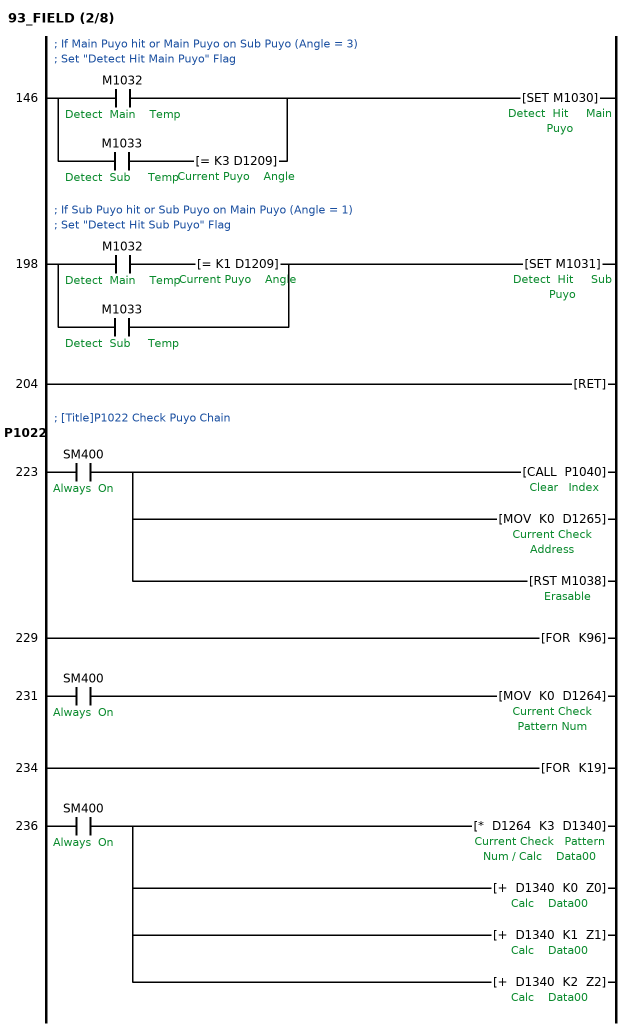
; If Main Puyo hit or Main Puyo on Sub Puyo (Angle = 3)
; Set "Detect Hit Main Puyo" Flag
146   LD      M1032  ; Detect  Main    Temp
      LD      M1033  ; Detect  Sub     Temp
      AND=    K3 D1209  ; Current Puyo    Angle
      ORB
      SET     M1030  ; Detect  Hit     Main    Puyo
; If Sub Puyo hit or Sub Puyo on Main Puyo (Angle = 1)
; Set "Detect Hit Sub Puyo" Flag
198   LD      M1032  ; Detect  Main    Temp
      AND=    K1 D1209  ; Current Puyo    Angle
      OR      M1033  ; Detect  Sub     Temp
      SET     M1031  ; Detect  Hit     Sub     Puyo
204   RET
; [Title]P1022 Check Puyo Chain
      P1022
223   LD      SM400  ; Always  On
      CALL    P1040
      MOV     K0 D1265  ; Current Check   Address
      RST     M1038  ; Erasable
229   FOR     K96
231   LD      SM400  ; Always  On
      MOV     K0 D1264  ; Current Check   Pattern Num
234   FOR     K19
236   LD      SM400  ; Always  On
      *       D1264 K3 D1340  ; Calc    Data00
      +       D1340 K0 Z0
      +       D1340 K1 Z1
      +       D1340 K2 Z2
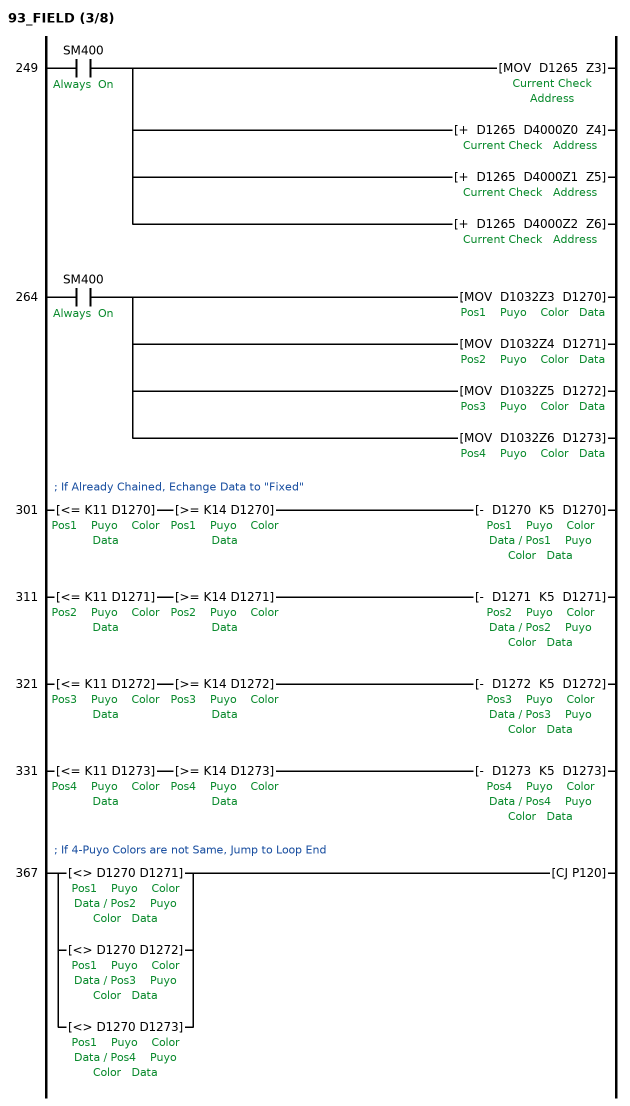
249   LD      SM400  ; Always  On
      MOV     D1265 Z3
      +       D1265 D4000Z0 Z4
      +       D1265 D4000Z1 Z5
      +       D1265 D4000Z2 Z6
264   LD      SM400  ; Always  On
      MOV     D1032Z3 D1270  ; Pos1    Puyo    Color   Data
      MOV     D1032Z4 D1271  ; Pos2    Puyo    Color   Data
      MOV     D1032Z5 D1272  ; Pos3    Puyo    Color   Data
      MOV     D1032Z6 D1273  ; Pos4    Puyo    Color   Data
; If Already Chained, Echange Data to "Fixed"
301   LD<=    K11 D1270  ; Pos1    Puyo    Color   Data
      AND>=   K14 D1270  ; Pos1    Puyo    Color   Data
      -       D1270 K5 D1270
311   LD<=    K11 D1271  ; Pos2    Puyo    Color   Data
      AND>=   K14 D1271  ; Pos2    Puyo    Color   Data
      -       D1271 K5 D1271
321   LD<=    K11 D1272  ; Pos3    Puyo    Color   Data
      AND>=   K14 D1272  ; Pos3    Puyo    Color   Data
      -       D1272 K5 D1272
331   LD<=    K11 D1273  ; Pos4    Puyo    Color   Data
      AND>=   K14 D1273  ; Pos4    Puyo    Color   Data
      -       D1273 K5 D1273
; If 4-Puyo Colors are not Same, Jump to Loop End
367   LD<>    D1270 D1271  ; Pos1    Puyo    Color   Data / Pos2    Puyo    Color   Data
      OR<>    D1270 D1272  ; Pos1    Puyo    Color   Data / Pos3    Puyo    Color   Data
      OR<>    D1270 D1273  ; Pos1    Puyo    Color   Data / Pos4    Puyo    Color   Data
      CJ      P120  ; Loop    End
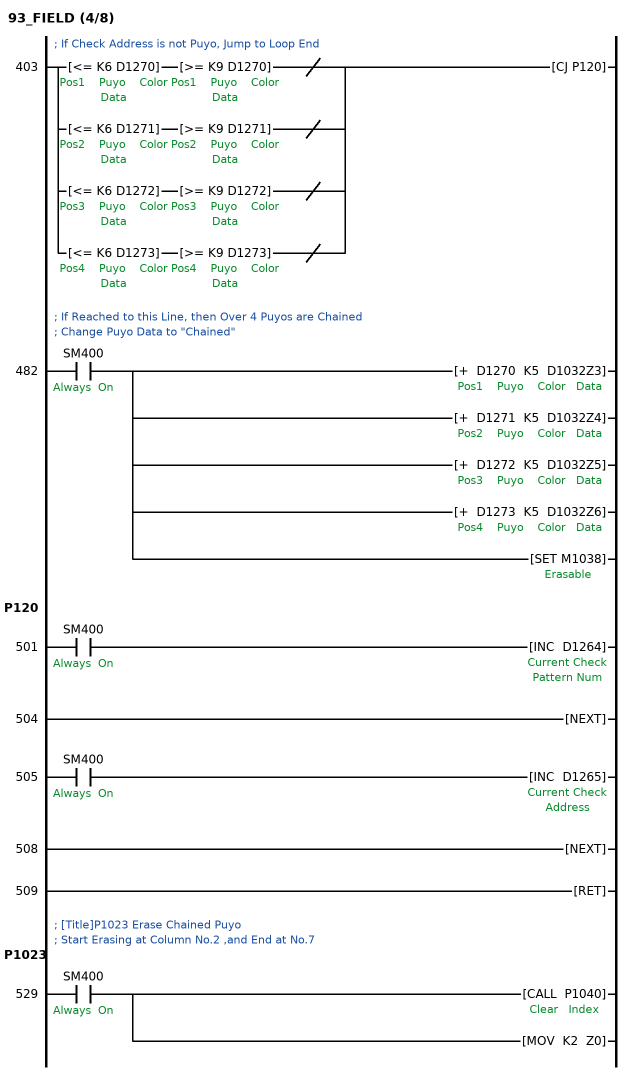
; If Check Address is not Puyo, Jump to Loop End
403   LD<=    K6 D1270  ; Pos1    Puyo    Color   Data
      AND>=   K9 D1270  ; Pos1    Puyo    Color   Data
      INV
      LD<=    K6 D1271  ; Pos2    Puyo    Color   Data
      AND>=   K9 D1271  ; Pos2    Puyo    Color   Data
      INV
      ORB
      LD<=    K6 D1272  ; Pos3    Puyo    Color   Data
      AND>=   K9 D1272  ; Pos3    Puyo    Color   Data
      INV
      ORB
      LD<=    K6 D1273  ; Pos4    Puyo    Color   Data
      AND>=   K9 D1273  ; Pos4    Puyo    Color   Data
      INV
      ORB
      CJ      P120
; If Reached to this Line, then Over 4 Puyos are Chained
; Change Puyo Data to "Chained"
482   LD      SM400  ; Always  On
      +       D1270 K5 D1032Z3
      +       D1271 K5 D1032Z4
      +       D1272 K5 D1032Z5
      +       D1273 K5 D1032Z6
      SET     M1038  ; Erasable
      P120
501   LD      SM400  ; Always  On
      INC     D1264
504   NEXT
505   LD      SM400  ; Always  On
      INC     D1265
508   NEXT
509   RET
; [Title]P1023 Erase Chained Puyo
      P1023
529   LD      SM400  ; Always  On
      CALL    P1040
      MOV     K2 Z0
